FUNCTION BYTES_TO_DWORD
  (* Standard: 61499-1; Description: Copyright (c) 2024 HR Agrartechnik GmbH This program and the accompanying materials are made available under the terms of the Eclipse Public License 2.0 which is available at https://www.eclipse.org/legal/epl-2.0/ SPDX-License-Identifier: EPL-2.0 *)
  (* Version 1.0, 2024-02-22, franz *)
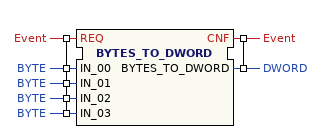
  EVENT_INPUT
    REQ WITH IN_00, IN_01, IN_02, IN_03;
  END_EVENT
  EVENT_OUTPUT
    CNF WITH BYTES_TO_DWORD;
  END_EVENT
  VAR_INPUT
    IN_00 : BYTE; (* BYTE 00 *)
    IN_01 : BYTE; (* BYTE 01 *)
    IN_02 : BYTE; (* BYTE 02 *)
    IN_03 : BYTE; (* BYTE 03 *)
  END_VAR
  VAR_OUTPUT
    BYTES_TO_DWORD : DWORD;
  END_VAR
  BODY IN ST:
FUNCTION BYTES_TO_DWORD : DWORD

VAR_INPUT
	IN_00 : BYTE;    // BYTE 00
	IN_01 : BYTE;    // BYTE 01
	IN_02 : BYTE;    // BYTE 02
	IN_03 : BYTE;    // BYTE 03
END_VAR

(* this Function combines the 2 BYTES to a word *)
BYTES_TO_DWORD := DWORD_BYTE_ZZ;
BYTES_TO_DWORD := BYTES_TO_DWORD OR SHL(BYTE_TO_DWORD(IN_03), SHFT_BYTE_03);
BYTES_TO_DWORD := BYTES_TO_DWORD OR SHL(BYTE_TO_DWORD(IN_02), SHFT_BYTE_02);
BYTES_TO_DWORD := BYTES_TO_DWORD OR SHL(BYTE_TO_DWORD(IN_01), SHFT_BYTE_01);
BYTES_TO_DWORD := BYTES_TO_DWORD OR SHL(BYTE_TO_DWORD(IN_00), SHFT_BYTE_00);

END_FUNCTION
  END_BODY
END_FUNCTION
